// TwinCAT 3 PLC project STS_04
// ProgramVersion: 3.1.4023.0
// libraries:
//   Tc2_Standard, * (Beckhoff Automation GmbH)
//   Tc2_System, * (Beckhoff Automation GmbH)
//   Tc3_Module, * (Beckhoff Automation GmbH)
//   TcUnit, * (www.tcunit.org)
// project tree:
//   DUTs/2. HMI/2.1 HMI Visualization/ dutVisuFeeder.TcDUT, dutVisuMain.TcDUT, dutVisuVBT.TcDUT, dutVisuEjection.TcDUT, dutVisuStacker.TcDUT
//   DUTs/3. Feeder/ FeederMode.TcDUT, FeederSimulation.TcDUT, FeedingState.TcDUT
//   DUTs/1. General State/ GeneralActiveProcessState.TcDUT, GeneralStateCommand.TcDUT, GeneralStateMain.TcDUT
//   DUTs/2. HMI/ HMI.TcDUT
//   DUTs/4. SheetAlignTable/ SheetAlignMode.TcDUT, SheetAlignState.TcDUT
//   DUTs/5. VacuumBeltTable/ VacuumBeltTableMode.TcDUT, VacuumBeltTableState.TcDUT
//   DUTs/6. EjectionGate/ EjectionGateMode.TcDUT, EjectionGateState.TcDUT
//   DUTs/7. StackerBeltTable/ StackerBeltTableMode.TcDUT, StackerBeltTableState.TcDUT
//   GVLs/ GVL.TcGVL, GVL_OOP.TcGVL
//   OOP/0. Program/ MAIN_OOP.TcPOU
//   OOP/1. Physical Buttons/Interface/ I_PB.TcIO
//   OOP/1. Physical Buttons/ PB_NOpen.TcPOU, PB_NClose.TcPOU
//   OOP/2. Physical Sensors/Interface/ I_Sensor.TcIO, O_Sensor.TcIO
//   OOP/2. Physical Sensors/ Sensor_NOpen.TcPOU, Sensor_NClose.TcPOU, Sensor_Trigger.TcPOU
//   OOP/5. Machine/0. Main Machine/ EjectionGate.TcPOU, Feeder.TcPOU, SAT.TcPOU, SBT.TcPOU, VBT.TcPOU
//   OOP/5. Machine/0. Main Machine/Interface/ MachineModule.TcIO
//   OOP/5. Machine/ P_MachineMain.TcPOU, STS.TcPOU
//   / PlcTask.TcTTO
//   POUs/0. FB/ Fb_AnalogToReal_Conversion.TcPOU, Fb_RealToAnalog_Conversion.TcPOU
//   POUs/1.2 Feeder Operation/ Fb_FeederOperation.TcPOU, Fb_FeedingStateCheck.TcPOU, P_Feeder.TcPOU
//   POUs/1.3 Sheet Align Table %28SAT%29/ P_SheetAlignTable.TcPOU (not stored)
//   POUs/1.4 Vacumm Belt Table %28VBT%29/ P_VacummBeltTable.TcPOU (not stored)
//   POUs/1.5 Ejection Gate/ P_EjectionGate.TcPOU
//   POUs/1.6 Stacker Belt Table %28SBT%29/ P_StackerBeltTable.TcPOU (not stored)
//   POUs/1.7 General Movement/ P_AllStateChecker.TcPOU, P_GeneralStateManager.TcPOU
//   POUs/ MAIN.TcPOU, P_Test.TcPOU
//   POUs_Test/ FB_Raw2Analog_Test.TcPOU, PRG_TEST.TcPOU
// real-time tasks:
//   TASK PlcTask: cycle T#10ms, priority 20, ADS port 350

CONFIGURATION STS_04
    RESOURCE PLC ON TwinCAT3
        TASK PlcTask(INTERVAL := T#10ms, PRIORITY := 20);
        PROGRAM MAIN WITH PlcTask : MAIN;
    END_RESOURCE
END_CONFIGURATION

// ---- DUTs/2. HMI/2.1 HMI Visualization/dutVisuFeeder.TcDUT
TYPE dutVisuFeeder :
STRUCT
	(*Values linked to HMI*)
	(*Feeder Operational values*)
	nFormatLength_mm   : INT;
	nSuctionLength_mm  : INT;
	nSheetGap_mm       : INT;
	tSingleSheetTime_s : INT;
	tCompilePostion_s  : INT;
	tDVPIDleOff_s      : INT;
	tDVPStartDelay_s   : INT;
	nMissingSheet      : INT;
	tApproachStop_s    : INT;
	
	(*Sheet Size Adjustment*)
	nSheetSize_mm		: INT;
	bSheetSizeIncrease  : BOOL;
	bSheetSizeDecrease  : BOOL;
	
	(*Feeder Movement setting*)
	bFeederUp			: BOOL;
	bFeederDown         : BOOL;

	(*Start Feeder*)	
	bStartFeeder		: BOOL;
	bStopFeeder			: BOOL;
END_STRUCT
END_TYPE

// ---- DUTs/2. HMI/2.1 HMI Visualization/dutVisuMain.TcDUT
TYPE dutVisuMain :
STRUCT
	(*Main Control*)
	bStartMachine			:BOOL;
	bStopMachine            :BOOL;
	bIncreaseMachineSpeed   :BOOL;
	bDecreaseMachineSpeed   :BOOL;
	                       
	nSheetCountAccepted     :INT;
	nSheetCountRejected     :INT;
	                        
	bSimulationMode         :BOOL;
END_STRUCT
END_TYPE

// ---- DUTs/2. HMI/2.1 HMI Visualization/dutVisuVBT.TcDUT
TYPE dutVisuVBT :
STRUCT
	
	(*Values linked to HMI*)
	(*Vacuum Belt Table Operational values*)
	nVmin_mMin  	: INT;
	nVmax_mMin		: INT;
	tStartDelay_s   : INT;
	tStopDelay_s 	: INT;
	bVisionBypass  	: INT;
	
	(*VBT Jogging*)
	bLeftJog		: BOOL;
	bRightJog  		: BOOL;
	nJogSpeed  		: INT;
	
	(*Fan Volume Control*)
	bFanIncrease	: BOOL;
	bFanDecrease    : BOOL;
	nFanSpeed_pct	: INT;

	(*Start Feeder*)	
	bStartFeeder	: BOOL;
	bStopFeeder		: BOOL;
	
END_STRUCT
END_TYPE

// ---- DUTs/2. HMI/2.1 HMI Visualization/dutVisuEjection.TcDUT
TYPE dutVisuEjection :
STRUCT
	(*Values linked to HMI*)
	(*Rejection Operation*)
	tDetectJamDuration_s	: INT;
	nBrakeDistance_mm		: INT;
	tBrakePulse_ms			: INT;

END_STRUCT
END_TYPE

// ---- DUTs/2. HMI/2.1 HMI Visualization/dutVisuStacker.TcDUT
TYPE dutVisuStacker :
STRUCT
	(*Values linked to HMI*)
	(*Stacker Operational values*)
	tOpenOscillator_s				: INT;
	tCloseJOgger_s      			: int;
	tDownBlas_ms        			: int;
	tDescentPulse_ms    			: int;
	                    			
	(*Stacker Plate Movement*)
	bStackerPlateUp					: BOOL;
	bStackerPlateDown   			: bool;
	                    			
	(*Alignment*)       	
	nAlignmentRation_n				: INT; (*ratio alignment, how many sheets has passed for alignment to trigger*)

	(*Brake Adjustment Control*)
	bIncreaseBrakeSpeedRatio		: BOOL;	
	bDecreaseBrakeSpeedRatio        : BOOL;
	nBrakeSpeedRatio                : INT;
	                                
	bIncreaseBrakeLength            : BOOL;
	bDecreaseBrakeLength            : BOOL;
	nBrakeSpeedLength               : INT;
	                               
	bIncreaseIntersheet             : BOOL;
	bDecreaseIntersheet	            : BOOL;
	nIntersheet                     : INT;

END_STRUCT
END_TYPE

// ---- DUTs/3. Feeder/FeederMode.TcDUT
{attribute 'qualified_only'}
{attribute 'strict'}
TYPE FeederMode :
(
	Mode_Jog		:= 0,
	Mode_Standard	:= 1,
	Mode_Simulation	:= 2
);
END_TYPE

// ---- DUTs/3. Feeder/FeederSimulation.TcDUT
TYPE FeederSimulation :
STRUCT
	i : INT;
END_STRUCT
END_TYPE

// ---- DUTs/3. Feeder/FeedingState.TcDUT
{attribute 'qualified_only'}
{attribute 'strict'}
TYPE FeedingState :
(
	State_Init 					,
	State_AutoStart         	,
	State_AutoHysterisis    	,
	State_AutoStop          	,
	State_AutoTopSensorReached 	,
	State_AutoFinalPosition     ,
	State_AutoBackToInit        ,
	State_Feeding				,
	State_Override				,
	State_Error					,
	State_ManualMoveUp			,
	State_ManualMoveDown    	
 
);
END_TYPE

// ---- DUTs/1. General State/GeneralActiveProcessState.TcDUT
TYPE GeneralActiveProcessState :
STRUCT
	FeederRunning				: BOOL;		 
	FeederStop                  : BOOL;
	FeederError                 : BOOL;
	                         
	SheetAlignTableRunning      : BOOL;
	SheetAlignTableStop         : BOOL;
	SheetAlignTableError        : BOOL;
END_STRUCT
END_TYPE

// ---- DUTs/1. General State/GeneralStateCommand.TcDUT
TYPE GeneralStateCommand :
STRUCT
	
	bStart		:BOOL;
	bStop       :BOOL;
	bOverride   :BOOL;
	bReset		:BOOL;
	
END_STRUCT
END_TYPE

// ---- DUTs/1. General State/GeneralStateMain.TcDUT
{attribute 'qualified_only'}
{attribute 'strict'}
TYPE GeneralStateMain :
(
	
	State_Init			,
	State_Reset         ,
	State_Run	        ,
	State_Stop          ,
	State_ErrorCheck       
);
END_TYPE

// ---- DUTs/2. HMI/HMI.TcDUT
TYPE HMI :
STRUCT
	//-----------------------------Auto----------------------------
	bAuto				:BOOL;
	bStart              :BOOL;
	bStop               :BOOL;
                        
	bFeederManualUp     :BOOL;
	bFeederManualDown   :BOOL;
	(*Visualization*)
	
	FeederOp			: dutVisuFeeder;
	VBTOp               : dutVisuVBT;
	EjectionOP          : dutVisuEjection;
	StackerOP           : dutVisuStacker;
	Main				: dutVisuMain;
	
END_STRUCT
END_TYPE

// ---- DUTs/4. SheetAlignTable/SheetAlignMode.TcDUT
{attribute 'qualified_only'}
{attribute 'strict'}
TYPE SheetAlignMode :
(
	Mode_Standard	:= 0,
	Mode_Manual		:= 1,
	Mode_Simulation	:= 2
	
);
END_TYPE

// ---- DUTs/4. SheetAlignTable/SheetAlignState.TcDUT
{attribute 'qualified_only'}
{attribute 'strict'}
TYPE SheetAlignState :
(
	State_Init 					,
	State_AutoStart         	,
	State_AutoStop          	,
	State_AutoBlowerOn			,
	State_AutoBackToInit        ,
	State_Override				,
	State_Error					
);
END_TYPE

// ---- DUTs/5. VacuumBeltTable/VacuumBeltTableMode.TcDUT
{attribute 'qualified_only'}
{attribute 'strict'}
TYPE VacuumBeltTableMode :
(
	Mode_Standard	:= 0,
	Mode_Manual		:= 1,
	Mode_Simulation	:= 2
	
);
END_TYPE

// ---- DUTs/5. VacuumBeltTable/VacuumBeltTableState.TcDUT
{attribute 'qualified_only'}
{attribute 'strict'}
TYPE VacuumBeltTableState :
(
	State_Init 					,
	State_AutoStart         	,
	State_AutoStop          	,
	State_AutoVacOn				,
	State_VacOff				,
	State_AutoBackToInit        ,
	State_Override				,
	State_Error					
);
END_TYPE

// ---- DUTs/6. EjectionGate/EjectionGateMode.TcDUT
{attribute 'qualified_only'}
{attribute 'strict'}
TYPE EjectionGateMode :
(
	Mode_Standard	:= 0,
	Mode_Manual		:= 1,
	Mode_Simulation	:= 2
	
);
END_TYPE

// ---- DUTs/6. EjectionGate/EjectionGateState.TcDUT
{attribute 'qualified_only'}
{attribute 'strict'}
TYPE EjectionGateState :
(
	State_Init 					,
	State_AutoStart         	,
	State_AutoStop          	,
	State_AutoEjectOn			,
	State_AutoBackToInit        ,
	State_Override				,
	State_Error					
);
END_TYPE

// ---- DUTs/7. StackerBeltTable/StackerBeltTableMode.TcDUT
{attribute 'qualified_only'}
{attribute 'strict'}
TYPE StackerBeltTableMode :
(
	Mode_Standard	:= 0,
	Mode_Manual		:= 1,
	Mode_Simulation	:= 2
	
);
END_TYPE

// ---- DUTs/7. StackerBeltTable/StackerBeltTableState.TcDUT
{attribute 'qualified_only'}
{attribute 'strict'}
TYPE StackerBeltTableState :
(
	State_Init 					,
	State_AutoStart         	,
	State_AutoStop          	,
	State_StackerStart			,
	State_StackerStop	        ,
	State_Override				,
	State_Error					
);
END_TYPE

// ---- GVLs/GVL.TcGVL
{attribute 'qualified_only'}
VAR_GLOBAL
	stHMI 		: HMI;
	stHMIsimul	: HMI;
	bHmiSimulation	: BOOL;
	
	stGSM : GeneralStateCommand; 
END_VAR

// ---- GVLs/GVL_OOP.TcGVL
{attribute 'qualified_only'}
VAR_GLOBAL
	//General Buttons
	(*Governs all things*)
	bStart 	: PB_NOpen; 
	bStop	: PB_NOpen;
	//bStart2 : PB_NClose;
	bEmergencyStop	:PB_NClose;
	
	(*sts component*)
	(*
		sts-feeder
		sts-sat
		sts-vbt
		sts-EjectGate
		sts-Stacker		
	*)
	(*sts-feeder*)
	bBottomHit 		: Sensor_NOpen;
	bTopHit			: Sensor_NOpen;
	bEnableFeeder	: Sensor_Trigger;	
	bUpFeeder		: Sensor_Trigger;
	bResetFeeder	: Sensor_Trigger;
	bDownFeeder     : Sensor_Trigger;
	nFeederTravel   : INT;
	
	(*Modules*)
	stHMI			: HMI;
	
	
	
	fbFeeder		: Feeder(bBottomHit,bTopHit);

	
	fbSTS : STS(bStart,
				bStop,
				bEmergencyStop,
				fbFeeder,
				stHMI);
	
(*OOP Logic*)	
(*
{Sensor Module}
		|
Integrated Into--->{Machine Module}
						|
					Integrated Into ---->{Main Machine}


*)
END_VAR

// ---- OOP/1. Physical Buttons/Interface/I_PB.TcIO
	INTERFACE I_PB

PROPERTY IsPressed : BOOL
//Property of PB when pressed
GET
END_GET
END_PROPERTY

PROPERTY IsReleased : BOOL
//Property of PB when is released
GET
END_GET
END_PROPERTY

END_INTERFACE

// ---- OOP/2. Physical Sensors/Interface/I_Sensor.TcIO
INTERFACE I_Sensor

PROPERTY isActive : BOOL
GET
END_GET
END_PROPERTY

END_INTERFACE

// ---- OOP/2. Physical Sensors/Interface/O_Sensor.TcIO
INTERFACE O_Sensor

PROPERTY isTriggered : BOOL
GET
END_GET
END_PROPERTY

END_INTERFACE

// ---- OOP/5. Machine/0. Main Machine/Interface/MachineModule.TcIO
INTERFACE MachineModule

METHOD Disable : BOOL
VAR_INPUT
END_VAR
END_METHOD

METHOD Enable : BOOL
VAR_INPUT
END_VAR
END_METHOD

METHOD Error : BOOL
VAR_INPUT
END_VAR
END_METHOD

METHOD Override : BOOL
VAR_INPUT
END_VAR
END_METHOD

METHOD Reset : BOOL
VAR_INPUT
END_VAR
END_METHOD

METHOD Start : BOOL
VAR_INPUT
END_VAR
END_METHOD

METHOD PUBLIC StateMachine
VAR_INPUT
END_VAR
END_METHOD

METHOD Stop : BOOL
VAR_INPUT
END_VAR
END_METHOD

END_INTERFACE

// ---- POUs/MAIN.TcPOU
PROGRAM MAIN
VAR
	fb_Test_Conversion : Fb_AnalogToReal_Conversion;
	ntest: LREAL;
	fb_testR2A: Fb_RealToAnalog_Conversion;
	stTestString : STRING :='Added this for 1.0.1';
END_VAR

P_Test();
P_Feeder();
P_SheetAlignTable();
P_VacummBeltTable();
P_EjectionGate();
P_StackerBeltTable();
P_AllStateChecker();
P_GeneralStateManager();
//PRG_TEST();

fb_Test_Conversion(iRawVal:= , iMinVal:=0 , iMaxVal:=180 , lActualVal=>ntest );
fb_testR2A(lActualVal:= , lMinVal:=50 , lMaxVal:=100 , iRawVal=> );

//OOP Test
MAIN_OOP();

END_PROGRAM

// ---- POUs/0. FB/Fb_AnalogToReal_Conversion.TcPOU
FUNCTION_BLOCK Fb_AnalogToReal_Conversion
VAR_INPUT
	iRawVal : UINT;
	iMinVal	: UINT;
	iMaxVal	: UINT;
	
END_VAR
VAR_OUTPUT
	lActualVal	: REAL;				//Actual converted value
	bError		: BOOL;
END_VAR           
VAR               
	lRangeHigh	: REAL := 32676;
	lRawVal 	: REAL;
	lMinVal		: REAL;
	lMaxVal		: REAL;
END_VAR

lRawVal	:=UINT_TO_REAL(iRawVal);
lMinVal	:=UINT_TO_REAL(iMinVal);
lMaxVal	:=UINT_TO_REAL(iMaxVal);

IF iRawVal<=0 THEN
	lActualVal:=0;
END_IF

IF NOT iRawVal>0 AND iRawVal<=lRangeHigh THEN	
	lActualVal := ((lMaxVal-lMinVal)/(lRangeHigh-0))*lRawVal+lMinVal;
	bError:=FALSE;
ELSE
	bError:=TRUE;	
END_IF

METHOD Error_Check : BOOL
VAR_INPUT
END_VAR
END_METHOD

METHOD RawToRealConversion : BOOL
VAR_INPUT
END_VAR
END_METHOD

END_FUNCTION_BLOCK

// ---- POUs/0. FB/Fb_RealToAnalog_Conversion.TcPOU
FUNCTION_BLOCK Fb_RealToAnalog_Conversion
VAR_INPUT
	lActualVal	: REAL;
	lMinVal		: REAL;
	lMaxVal		: REAL;
	
END_VAR
VAR_OUTPUT
	iRawVal	: UINT;					//Raw converted sensor values
END_VAR           
VAR               
	lRangeHigh	: REAL := 32676;
	lRawVal : REAL;

END_VAR


IF lActualVal <=0 THEN
	iRawVal:=0;
END_IF

IF lActualVal>0 THEN
	lRawVal:=(lActualVal-lMinVal)*((lRangeHigh-0)/(lMaxVal-lMinVal));
END_IF

END_FUNCTION_BLOCK

// ---- POUs/P_Test.TcPOU
PROGRAM P_Test
VAR
	
nAngle : LREAL;
nAngle_decimal : int;
nAngle_Final : LREAL;
sWriteFromHMI : STRING;
sWriteToHMI : STRING:='This Is From PLC';
b_HMI_StartLine : BOOL;
b_HMI_StopLine : BOOL;
bStartTrig: R_TRIG;
bStopTrig: R_TRIG;

bSpeedInc		:BOOL;
bSpeedDecrease  :BOOL;
stStatus		:STRING;
// State
n : INT;
END_VAR


bStartTrig(CLK:=b_HMI_StartLine , Q=> );
bStopTrig(CLK:=b_HMI_StopLine , Q=> );

IF ( stStatus='' OR stStatus='Stopped') 
	AND bStartTrig.Q THEN
	stStatus:='Started';

END_IF

IF stStatus='Started' AND bStopTrig.Q THEN
	stStatus:='Stopped';
	nAngle :=0;
END_IF

IF  stStatus='Started' THEN
	
	IF nAngle<180 THEN
		nAngle :=nAngle+0.01;
	END_IF
	//nAngle_decimal:=find((LREAL_TO_STRING(nAngle)),'.');
		
	IF nAngle>=180 THEN
		nAngle :=0;
	END_IF
END_IF
nAngle_Final :=LREAL_TO_UINT(STRING_TO_LREAL(left((LREAL_TO_STRING(nAngle)),((find((LREAL_TO_STRING(nAngle)),'.'))+2))));

END_PROGRAM

// ---- POUs/1.2 Feeder Operation/P_Feeder.TcPOU
PROGRAM P_Feeder
VAR
	bStartFeeder : BOOL;
	bFeederOK: BOOL;
	//dut_FeedingState : FeedingState;
	fbFb_FeedingStateCheck: Fb_FeedingStateCheck;	
//-----------------------------------Feeder Mode -------------------------//
	iFeederMode : INT;	
	bGoCounter, bSetCounter AT %Q*:BOOL;
	wFrequencyValue, wTargetCounterValue, wSetCounterValue AT %Q*:WORD;
	wCounterValue AT %I*:WORD;
	nState, nCntCycle:UDINT;
	bStart:BOOL;
	wFrequencyValue_Test:WORD:=200;
	nPrevValue			:WORD;
	wTargetCounterValue_Test:WORD:=180;
	bHitTop : BOOL;
	bHitBottom : BOOL;
	bTargetDistanceHitUP	: BOOL;
	bTargetDistanceHitDown	: BOOL;

//------------------------------------CASE-------------------------------//
	ifeedercase : INT;

(* For reference
	State_Init 					:= 1,
	State_AutoStart         	:= 2,
	State_AutoHysterisis    	:= 3,
	State_AutoStop          	:= 4,
	State_AutoTopSensorReached 	:= 5,
	State_AutoFinalPosition     := 6,
	State_AutoBackToInit        := 7,
	State_Feeding				:= 8,
	State_Override				:= 9,
	State_Error					:= 10,
	State_ManualMoveUp			:= 11,
	State_ManualMoveDown    	:= 12
*)	
//-------------------------Simulated Values-----------------------------//
nCurrentValue 	: DWORD;
nTargetValue	: DWORD;
	
END_VAR
VAR_INPUT
	bStartCommand : BOOL;
END_VAR

IF GVL.bHmiSimulation THEN
	GVL.stHMIsimul:=GVL.stHMI;
	iFeederMode:=FeederMode.Mode_Simulation;
END_IF 
IF NOT GVL.bHmiSimulation THEN
	GVL.stHMI:=GVL.stHMI;
	iFeederMode:=FeederMode.Mode_Standard;
END_IF

CASE ifeedercase OF

FeedingState.State_Init 			:	//Awaiting for command   
	IF GVL.stHMI.bAuto  THEN
		ifeedercase:=FeedingState.State_AutoStart;
	END_IF
	IF GVL.stHMI.bFeederManualDown THEN
		ifeedercase:=FeedingState.State_ManualMoveDown;	
	END_IF
	IF GVL.stHMI.bFeederManualUp THEN
		ifeedercase:=FeedingState.State_ManualMoveUp;
	END_IF	
	IF NOT (iFeederMode=FeederMode.Mode_Simulation) THEN // go back to init
		iFeederCase:=FeedingState.State_Init;
		wTargetCounterValue:=0;
		nPrevValue:=0;	
		bHitTop:=FALSE;	
		bHitBottom:=FALSE;
		bTargetDistanceHitUp:=FALSE;
		bTargetDistanceHitDown:=FALSE;
		nState:=0;
	END_IF
	
FeedingState.State_AutoStart            : 	//Start 

	IF NOT bStartFeeder THEN
		ifeedercase:= FeedingState.State_AutoBackToInit;
	END_IF
	IF GVL.bHmiSimulation THEN
		//Adding Feeder movement simulation
		;
	END_IF
FeedingState.State_AutoHysterisis       : 
FeedingState.State_AutoStop             : 
FeedingState.State_AutoTopSensorReached :	
FeedingState.State_AutoFinalPosition    : 
FeedingState.State_AutoBackToInit       : 
FeedingState.State_Feeding				:        
FeedingState.State_Override				:       
FeedingState.State_Error				:	
     
FeedingState.State_ManualMoveUp			:
	IF iFeederMode=FeederMode.Mode_Simulation THEN
		CASE nState OF
				0: //Check ongoing or Initial Start
					IF gvl.stHMI.bFeederManualUp THEN
						IF NOT (bHitTop OR bTargetDistanceHitUp) THEN
							IF nPrevValue=0 
							AND wTargetCounterValue=0 THEN // Coming from initialization
								nState:=20;
							END_IF
							IF wTargetCounterValue>nPrevValue THEN //Continuation
								nPrevValue:=wTargetCounterValue;
								nState:=20;
							END_IF
						ELSE
							nState:=0;
							nPrevValue:=wTargetCounterValue;
						END_IF
					END_IF	
					
				20://Increment and making sure previous values are recorded.			
							IF (wTargetCounterValue>nPrevValue) THEN
								nState:=30;
							END_IF
							IF (wTargetCounterValue=nPrevValue) THEN
								wTargetCounterValue:=wTargetCounterValue+1;
								nState:=20;
							END_IF

				30:	//Check if reached target or not
					IF wTargetCounterValue < wTargetCounterValue_Test THEN //not reached
						nstate:=0;
					END_IF
					IF wTargetCounterValue >= wTargetCounterValue_Test OR bHitTop THEN // Reached sensor top or movement set
						nState:=40;
					END_IF
				40:	
					nState:=0;
					bTargetDistanceHitUp:=TRUE;
					bFeederOK :=TRUE;
					
				
		END_CASE
	END_IF
	IF iFeederMode=FeederMode.Mode_Jog THEN
		;
	END_IF
	ifeedercase:= FeedingState.State_Init;
	
FeedingState.State_ManualMoveDown		:
	IF iFeederMode=FeederMode.Mode_Simulation THEN
		CASE nState OF
				0: //Check ongoing or Initial Start
					IF gvl.stHMI.bFeederManualDown THEN
						IF NOT (bHitBottom OR bTargetDistanceHitDown) THEN
							IF nPrevValue=0 
							AND wTargetCounterValue=0 THEN // Coming from initialization
								nState:=20;
							END_IF
							IF wTargetCounterValue>nPrevValue THEN //Continuation
								nPrevValue:=wTargetCounterValue;
								nState:=20;
							END_IF
						ELSE
							nState:=0;
							nPrevValue:=wTargetCounterValue;
						END_IF
					END_IF	
					
				20://Increment and making sure previous values are recorded.			
							IF (wTargetCounterValue>nPrevValue) THEN
								nState:=30;
							END_IF
							IF (wTargetCounterValue=nPrevValue) THEN
								wTargetCounterValue:=wTargetCounterValue+1;
								nState:=20;
							END_IF

				30:	//Check if reached target or not
					IF wTargetCounterValue < wTargetCounterValue_Test THEN //not reached
						nstate:=0;
					END_IF
					IF wTargetCounterValue >= wTargetCounterValue_Test OR bHitTop THEN // Reached sensor top or movement set
						nState:=40;
					END_IF
				40:	
					nState:=0;
					bTargetDistanceHitDown:=TRUE;
				
		END_CASE
	END_IF
	IF iFeederMode=FeederMode.Mode_Jog THEN
		;
	END_IF
	ifeedercase:= FeedingState.State_Init;
	

END_CASE

END_PROGRAM

// ---- POUs/1.2 Feeder Operation/Fb_FeedingStateCheck.TcPOU
FUNCTION_BLOCK Fb_FeedingStateCheck
VAR_INPUT
	dut_FeedingState : FeedingState;
END_VAR
VAR_OUTPUT
	iReadableFeedingState : INT; // number which represent the state
END_VAR
VAR
	iBareNum : INT; // number we use to cycle through the FeedingState
	iLastFeedingState : FeedingState;
	
	nCaseNumberCycler : INT;
END_VAR

CASE nCaseNumberCycler OF
0: //Check if number is 0 or not. As 0 would represent initialized state
	//Also check whether it is there are any state changes or not
	IF (dut_FeedingState = iLastFeedingState ) THEN
		nCaseNumberCycler:=0;
	ELSE
		nCaseNumberCycler:=10;
	END_IF
	
10: //Cycling
	FOR iBareNum:=0 TO 11 BY 1 DO
		IF iBareNum < dut_FeedingState THEN
			iBareNum:=iBareNum+1;
		END_IF
		IF iBareNum > dut_FeedingState THEN
			iBareNum:=iBareNum-1;
		END_IF
		
	END_FOR
nCaseNumberCycler:=50;
50:	
nCaseNumberCycler:=0;
END_CASE

END_FUNCTION_BLOCK

// ---- POUs/1.5 Ejection Gate/P_EjectionGate.TcPOU
PROGRAM P_EjectionGate
VAR
		(*Initialization*)
	bEJ_OK		: BOOL;
	bError		: BOOL;
	bStart		: BOOL;
	bStop		: BOOL;
	(*Process*)
	bEjEnable 	: BOOL;
	bEjectOn	: BOOL;
	bEjectOff	: BOOL;
	bOverride	: BOOL;
	(*Ejection Gate Specific Process*)
	bSheetStuck		: BOOL;
	bSheetPresence		: BOOL;
	nSheetCount		: INT;
	FB_SheetCount_Trig	: R_TRIG;
	tSheetStuck_s	: TIME :=T#5S ;
	
	
	//-----------------------------------------(*Case*)-----------------------------------------------------
	
	(* Reference for VBT

	State_Init 					,
	State_AutoStart         	,
	State_AutoStop          	,
	State_AutoEjectOn			,
	State_AutoBackToInit        ,
	State_Override				,
	State_Error			
	*)	
	
	asd: R_TRIG;
	FbSheetStuckCheck: TON;
END_VAR
VAR_INPUT
	bStartCommand : BOOL;
END_VAR
VAR_OUTPUT
	iEJcase : INT;
END_VAR

CASE iEJcase OF
EjectionGateState.State_Init			:	

	IF (bEJ_OK AND bStartCommand)  
	AND NOT bError THEN
		iEJcase:= EjectionGateState.State_AutoStart;
	END_IF 
	IF bError THEN
		iEJcase:= EjectionGateState.State_Error;
	END_IF

   
EjectionGateState.State_AutoStart     	:
	IF bStop THEN
		iEJcase:= EjectionGateState.State_AutoStop;
	ELSE
		iEJcase :=EjectionGateState.State_AutoEjectOn;
	END_IF


EjectionGateState.State_AutoStop      	:
	iEJcase:= EjectionGateState.State_AutoBackToInit;


EjectionGateState.State_AutoEjectOn	  	:
	(*Insert business logic here*)
	(*Ejection*)
	IF P_VacummBeltTable.bBadSheetSignal THEN
		bEjectOn :=TRUE;
	END_IF // Need to add business logic to count for speed/time on-site.
	
	(*Sheet Counting*)
	FB_SheetCount_Trig(CLK:= bSheetPresence, Q=> );
	IF FB_SheetCount_Trig.Q THEN
		nSheetCount:=nSheetCount+1;
	END_IF
	FbSheetStuckCheck(IN:=bSheetPresence , PT:=tSheetStuck_s , Q=> , ET=> );
	IF FbSheetStuckCheck.Q THEN
		bSheetStuck:=TRUE;
		iEJcase:= EjectionGateState.State_Error;
	END_IF


EjectionGateState.State_AutoBackToInit	:
	iEJcase:= EjectionGateState.State_Init;


EjectionGateState.State_Override		:   
	;


EjectionGateState.State_Error			:     
	IF bError THEN
		iEJcase:= EjectionGateState.State_AutoBackToInit;
	END_IF

END_CASE

END_PROGRAM

// ---- POUs/1.7 General Movement/P_AllStateChecker.TcPOU
PROGRAM P_AllStateChecker
VAR
	(*
		Author - Gideon Jgordon (GJ)
		Changes 
		-(GJ) stGSM moved here
	*)	
	bAllOk : BOOL;	// All OK process
	//bSAT_OK: BOOL;  //SAT Process OK
END_VAR


IF P_GeneralStateManager.nStateGeneral =GeneralStateMain.State_ErrorCheck THEN
	gvl.stGSM.bStop			:=TRUE;
	gvl.stGSM.bOverride		:=FALSE;
	gvl.stGSM.bStart		:=FALSE;
	gvl.stGSM.bReset		:=TRUE;	
END_IF

IF P_GeneralStateManager.nStateGeneral =GeneralStateMain.State_Init THEN
	gvl.stGSM.bStop		   :=TRUE;
	gvl.stGSM.bOverride	   :=TRUE;
	gvl.stGSM.bStart	   :=FALSE;
	gvl.stGSM.bReset	   :=FALSE;	
END_IF

IF P_GeneralStateManager.nStateGeneral =GeneralStateMain.State_Reset THEN
	gvl.stGSM.bStop		   :=TRUE;
	gvl.stGSM.bOverride	   :=FALSE;
	gvl.stGSM.bStart	   :=FALSE;
	gvl.stGSM.bReset	   :=TRUE;	
END_IF

IF P_GeneralStateManager.nStateGeneral =GeneralStateMain.State_Run THEN
	gvl.stGSM.bStop		   :=TRUE;
	gvl.stGSM.bOverride	   :=FALSE;
	gvl.stGSM.bStart	   :=FALSE;
	gvl.stGSM.bReset	   :=FALSE;
END_IF

IF P_GeneralStateManager.nStateGeneral =GeneralStateMain.State_Stop THEN
	gvl.stGSM.bStop		   :=TRUE;
	gvl.stGSM.bOverride	   :=FALSE;
	gvl.stGSM.bStart	   :=FALSE;
	gvl.stGSM.bReset	   :=FALSE;
END_IF

IF  	P_Feeder.bFeederOK 
	AND P_SheetAlignTable.bSAT_OK 
	AND P_VacummBeltTable.bVBT_OK
	AND P_EjectionGate.bEJ_OK
	AND P_StackerBeltTable.bSBT_OK		THEN
	bAllok:=TRUE;
ELSE
	bAllok:=FALSE;	
END_IF

END_PROGRAM

// ---- POUs/1.7 General Movement/P_GeneralStateManager.TcPOU
PROGRAM P_GeneralStateManager
VAR
	(*
		Author - Gideon Jgordon (GJ)
		Changes 
		-(GJ) Added to govern the General State of the STS04 Machine 
		-(GJ) stGSM moved to P_AllStateChecker to make it cleaner
	*)	
	nStateGeneral : INT;
	bValuesResetDone: BOOL;
END_VAR

CASE nStateGeneral OF

GeneralStateMain.State_Init				: //Initialize all the state

	IF gvl.stHMI.bStart THEN
		nStateGeneral:= GeneralStateMain.State_Reset;
		ELSE
		nStateGeneral:=	GeneralStateMain.State_Init;
	END_IF	
	
GeneralStateMain.State_Reset			: // Reset behaviour and values befor we proceed to go into Run Mode

	//Adding reset below here
	IF (bValuesResetDone AND P_AllStateChecker.bAllOk) THEN
		nStateGeneral:=GeneralStateMain.State_Run;
		gvl.stGSM.bStart	:=TRUE;
	END_IF
	IF NOT (bValuesResetDone AND P_AllStateChecker.bAllOk) THEN
		nStateGeneral:=GeneralStateMain.State_Init;
	END_IF
	
GeneralStateMain.State_Run              : // Governs the Process during run

	IF NOT P_AllStateChecker.bAllOk THEN
		gvl.stGSM.bStart	:=FALSE;
	END_IF
	IF gvl.stHMI.bStop THEN
		nStateGeneral:= GeneralStateMain.State_Stop;
		gvl.stGSM.bStart	:=FALSE;
	END_IF
	
GeneralStateMain.State_Stop             : //Stop via HMI or Error

	nStateGeneral:= GeneralStateMain.State_Init;
	
GeneralStateMain.State_ErrorCheck       :

	
	
END_CASE

END_PROGRAM

// ---- OOP/0. Program/MAIN_OOP.TcPOU
PROGRAM MAIN_OOP
VAR
	bStartButton : PB_NOpen;
	bStopButton :PB_NOpen;
	bEstopButton : PB_NClose;
	bProcessStart : BOOL;
	bProcessError : BOOL;
	bProcessOverride : BOOL;
	
	//Feeder
	bStartFeeder		: BOOL;
	bStopFeeder			: BOOL;
	bFeederError        : BOOL;
	                   
	bFeederAuto         : BOOL;
	bFeederUpAuto       : BOOL;
	bFeederDownAuto     : BOOL;
	                   
	bFeederManual       : BOOL;
	bFeederUpManual     : BOOL;
	bFeederDownManual   : BOOL;
	
	bFeederAtPos		: BOOL;
	
	// SAT
	
	
END_VAR

IF bStartButton.IsPressed AND bStopButton.IsPressed THEN
	bStartFeeder:=TRUE;
END_IF
IF bStopButton.IsPressed AND bStartButton.IsPressed THEN
	bStopFeeder :=FALSE;
END_IF

P_MachineMain();

END_PROGRAM

// ---- OOP/1. Physical Buttons/PB_NOpen.TcPOU
FUNCTION_BLOCK PB_NOpen IMPLEMENTS I_PB
VAR
	bInput AT %I* :BOOL;
	
END_VAR

PROPERTY IsPressed : BOOL
//Property of PB when pressed
GET
VAR
	//Giving the properties of bInputSensor to isPressed
END_VAR
IsPressed := bInput;
END_GET
END_PROPERTY

PROPERTY IsReleased : BOOL
//Property of PB when PBNOpen is released
GET
VAR
	//Giving the properties of bInputSensor to isPressed
END_VAR
IsReleased := NOT bInput;
END_GET
END_PROPERTY

END_FUNCTION_BLOCK

// ---- OOP/1. Physical Buttons/PB_NClose.TcPOU
FUNCTION_BLOCK PB_NClose IMPLEMENTS I_PB
VAR
	bInput AT %I* :BOOL;
	
END_VAR

PROPERTY IsPressed : BOOL
// Property of PB button when it is pressed but for normally close
GET
IsPressed := NOT bInput;
END_GET
END_PROPERTY

PROPERTY IsReleased : BOOL
// Property of PB button when it is Released State but for normally close
GET
IsReleased := bInput;
END_GET
END_PROPERTY

END_FUNCTION_BLOCK

// ---- OOP/5. Machine/P_MachineMain.TcPOU
PROGRAM P_MachineMain
VAR
	
END_VAR

GVL_OOP.fbFeeder();
GVL_OOP.fbSTS();

END_PROGRAM

// ---- OOP/5. Machine/STS.TcPOU
FUNCTION_BLOCK STS
VAR
	bStart	: I_PB; // ref this to NO How to reference this as NO or NC????
	//bStart2	: I_PB;
	bStop	: I_PB; // ref this of NO
	bEmergency	: I_PB; // ref this to NC
	Feeder : MachineModule; // ref this to MachineModule
	
	// HMI here
	STS_Hmi : HMI;	
	
	

END_VAR

IF bStart.IsPressed AND bStop.IsReleased THEN
	Feeder.Enable();
END_IF

IF bStart.IsReleased AND bStop.IsPressed THEN
	Feeder.Disable();
END_IF

IF bEmergency.IsPressed THEN
	Feeder.Disable();
END_IF

METHOD FB_init : BOOL
VAR_INPUT
	bInitRetains : BOOL; // if TRUE, the retain variables are initialized (warm start / cold start)
	bInCopyCode : BOOL;  // if TRUE, the instance afterwards gets moved into the copy code (online change)
	
// Parsing it so that the STS declared need to have 4 arguments	
	bStart	: I_PB; // ref this to NO How to reference this as NO or NC????
	bStop	: I_PB; // ref this of NO
	bEmergency	: I_PB; // ref this to NC
	
	//Machine Modules
	Feeder : MachineModule; // ref this to MachineModule
	STS_Hmi : HMI;	
	
END_VAR
THIS^.bStart			:= bStart;
THIS^.bStop			:= bStop;
THIS^.bEmergency	    := bEmergency;
THIS^.Feeder          := Feeder;
THIS^.STS_Hmi         := STS_Hmi;
END_METHOD

END_FUNCTION_BLOCK

// ---- OOP/5. Machine/0. Main Machine/Feeder.TcPOU
FUNCTION_BLOCK Feeder IMPLEMENTS MachineModule
VAR
	(*General Movement Trigger*)
	bEnable			: BOOL;
	bDisable        : BOOL;
	bError          : BOOL;
	bOverride       : BOOL;
	bSimulation     : BOOL;
	bStart          : BOOL;
	bStop           : BOOL;
	
	(*Sensor Specific Trigger*)
	bBottomHit 		: I_Sensor;
	bTopHit			: I_Sensor;
	(*Internal Variable*)
	nMovement 		: INT;
	nmovetest		: INT;
	(*Fedder*)
	bFeederPlateInPos	: BOOL;

END_VAR

(*Business Logic here*)

IF 	bEnable 
	AND NOT (bError)
	AND nMovement<1500 THEN
	
	nMovement := nMovement+1;
	bStop:=FALSE; (*Could use this thing in another module*)
	
END_IF

IF nMovement=1500 THEN
	bStop:=TRUE;
END_IF

METHOD Disable : BOOL 
VAR_INPUT
END_VAR
bEnable:=FALSE;
END_METHOD

METHOD Enable : BOOL
VAR_INPUT
END_VAR
bEnable:=TRUE;
bDisable:=FALSE;
END_METHOD

METHOD Error : BOOL
VAR_INPUT
END_VAR
bEnable:=FALSE;
END_METHOD

METHOD FB_init : BOOL
VAR_INPUT
	bInitRetains : BOOL; // if TRUE, the retain variables are initialized (warm start / cold start)
	bInCopyCode : BOOL;  // if TRUE, the instance afterwards gets moved into the copy code (online change)
	bBottomHit 		: I_Sensor;
	bTopHit			: I_Sensor;
END_VAR
THIS^.bBottomHit	:= bBottomHit;
THIS^.bTopHit		:= bTopHit;
END_METHOD

METHOD Override : BOOL
VAR_INPUT
END_VAR
END_METHOD

METHOD Reset : BOOL
VAR_INPUT
END_VAR
END_METHOD

METHOD Start : BOOL
VAR_INPUT
END_VAR
END_METHOD

METHOD PUBLIC StateMachine
VAR_INPUT

END_VAR
IF bEnable THEN
	nmovetest:=nmovetest+1;	
	ELSE
		
	nmovetest:=0;
END_IF
END_METHOD

METHOD Stop : BOOL
VAR_INPUT
END_VAR
END_METHOD

END_FUNCTION_BLOCK

// ---- OOP/5. Machine/0. Main Machine/SAT.TcPOU
FUNCTION_BLOCK SAT IMPLEMENTS MachineModule
VAR
	bEnable			: BOOL;
	bDisable        : BOOL;
	bError          : BOOL;
	bOverride       : BOOL;
	bSimulation     : BOOL;
	bStart          : BOOL;
	bStop           : BOOL;
END_VAR

// This is the core module needed that we are creating for our STS and contains everything related to the STS

// To be added
(*
FEEDER

SAT

VBT

EJECT

GATE

SBT

*)

METHOD Disable : BOOL
VAR_INPUT
END_VAR
bEnable:=FALSE;
END_METHOD

METHOD Enable : BOOL
VAR_INPUT
END_VAR
bEnable:=TRUE;
bDisable:=False;
END_METHOD

METHOD Error : BOOL
VAR_INPUT
END_VAR
bEnable:=FALSE;
END_METHOD

METHOD Override : BOOL
VAR_INPUT
END_VAR
END_METHOD

METHOD Reset : BOOL
VAR_INPUT
END_VAR
END_METHOD

METHOD Start : BOOL
VAR_INPUT
END_VAR
END_METHOD

METHOD PUBLIC StateMachine
VAR_INPUT
END_VAR
END_METHOD

METHOD Stop : BOOL
VAR_INPUT
END_VAR
END_METHOD

END_FUNCTION_BLOCK

// ---- OOP/5. Machine/0. Main Machine/VBT.TcPOU
FUNCTION_BLOCK VBT IMPLEMENTS MachineModule
VAR
	bEnable			: BOOL;
	bDisable        : BOOL;
	bError          : BOOL;
	bOverride       : BOOL;
	bSimulation     : BOOL;
	bStart          : BOOL;
	bStop           : BOOL;
END_VAR

// This is the core module needed that we are creating for our STS and contains everything related to the STS

// To be added
(*
FEEDER

SAT

VBT

EJECT

GATE

SBT

*)

METHOD Disable : BOOL
VAR_INPUT
END_VAR
bEnable:=FALSE;
END_METHOD

METHOD Enable : BOOL
VAR_INPUT
END_VAR
bEnable:=TRUE;
bDisable:=False;
END_METHOD

METHOD Error : BOOL
VAR_INPUT
END_VAR
bEnable:=FALSE;
END_METHOD

METHOD Override : BOOL
VAR_INPUT
END_VAR
END_METHOD

METHOD Start : BOOL
VAR_INPUT
END_VAR
END_METHOD

METHOD PUBLIC StateMachine
VAR_INPUT
END_VAR
END_METHOD

METHOD Stop : BOOL
VAR_INPUT
END_VAR
END_METHOD

END_FUNCTION_BLOCK

// ---- OOP/2. Physical Sensors/Sensor_NOpen.TcPOU
FUNCTION_BLOCK Sensor_NOpen IMPLEMENTS I_Sensor
VAR
	bInput AT %I* : BOOL;
END_VAR

PROPERTY isActive : BOOL
GET
isActive:=bInput;
END_GET
END_PROPERTY

PROPERTY notActive : BOOL
GET
notActive:= NOT bInput;
END_GET
END_PROPERTY

END_FUNCTION_BLOCK

// ---- OOP/2. Physical Sensors/Sensor_Trigger.TcPOU
FUNCTION_BLOCK Sensor_Trigger implements O_Sensor
VAR
	bOutput AT %Q* : BOOL;
END_VAR

PROPERTY isTriggered : BOOL
GET
isTriggered:=bOutput;
END_GET
END_PROPERTY

END_FUNCTION_BLOCK

// ---- OOP/2. Physical Sensors/Sensor_NClose.TcPOU
FUNCTION_BLOCK Sensor_NClose IMPLEMENTS I_Sensor
VAR
	bInput AT %I* : BOOL;
END_VAR

PROPERTY isActive : BOOL
GET
isActive:= not bInput;
END_GET
END_PROPERTY

PROPERTY notActive : BOOL
GET
isActive := bInput;
END_GET
END_PROPERTY

END_FUNCTION_BLOCK

// ---- OOP/5. Machine/0. Main Machine/EjectionGate.TcPOU
FUNCTION_BLOCK EjectionGate IMPLEMENTS MachineModule
VAR
	bEnable			: BOOL;
	bDisable        : BOOL;
	bError          : BOOL;
	bOverride       : BOOL;
	bSimulation     : BOOL;
	bStart          : BOOL;
	bStop           : BOOL;
END_VAR

// This is the core module needed that we are creating for our STS and contains everything related to the STS

// To be added
(*
FEEDER

SAT

VBT

EJECT

GATE

SBT

*)

METHOD Disable : BOOL
VAR_INPUT
END_VAR
bEnable:=FALSE;
END_METHOD

METHOD Enable : BOOL
VAR_INPUT
END_VAR
bEnable:=TRUE;
bDisable:=False;
END_METHOD

METHOD Error : BOOL
VAR_INPUT
END_VAR
bEnable:=FALSE;
END_METHOD

METHOD Override : BOOL
VAR_INPUT
END_VAR
END_METHOD

METHOD Reset : BOOL
VAR_INPUT
END_VAR
END_METHOD

METHOD Start : BOOL
VAR_INPUT
END_VAR
END_METHOD

METHOD PUBLIC StateMachine
VAR_INPUT
END_VAR
END_METHOD

METHOD Stop : BOOL
VAR_INPUT
END_VAR
END_METHOD

END_FUNCTION_BLOCK

// ---- OOP/5. Machine/0. Main Machine/SBT.TcPOU
FUNCTION_BLOCK SBT IMPLEMENTS MachineModule
VAR
	bEnable			: BOOL;
	bDisable        : BOOL;
	bError          : BOOL;
	bOverride       : BOOL;
	bSimulation     : BOOL;
	bStart          : BOOL;
	bStop           : BOOL;
END_VAR

// This is the core module needed that we are creating for our STS and contains everything related to the STS

// To be added
(*
FEEDER

SAT

VBT

EJECT

GATE

SBT

*)

METHOD Disable : BOOL
VAR_INPUT
END_VAR
bEnable:=FALSE;
END_METHOD

METHOD Enable : BOOL
VAR_INPUT
END_VAR
bEnable:=TRUE;
bDisable:=False;
END_METHOD

METHOD Error : BOOL
VAR_INPUT
END_VAR
bEnable:=FALSE;
END_METHOD

METHOD Override : BOOL
VAR_INPUT
END_VAR
END_METHOD

METHOD Reset : BOOL
VAR_INPUT
END_VAR
END_METHOD

METHOD Start : BOOL
VAR_INPUT
END_VAR
END_METHOD

METHOD PUBLIC StateMachine
VAR_INPUT
END_VAR
END_METHOD

METHOD Stop : BOOL
VAR_INPUT
END_VAR
END_METHOD

END_FUNCTION_BLOCK

// ---- POUs/1.2 Feeder Operation/Fb_FeederOperation.TcPOU
FUNCTION_BLOCK Fb_FeederOperation
VAR_INPUT
	nModeSelector	: FeederMode;
	bEnable         : BOOL;
END_VAR
VAR_OUTPUT
	bJogFwd         : BOOL;
	bJogRev         : BOOL;
END_VAR
VAR
END_VAR

;

END_FUNCTION_BLOCK

// ---- POUs_Test/FB_Raw2Analog_Test.TcPOU
FUNCTION_BLOCK FB_Raw2Analog_Test extends FB_TestSuite
VAR
END_VAR

TestRawVal2RealValConversion();

METHOD PRIVATE TestRawVal2RealValConversion EXTENDS FB_TestSuite
VAR
	Fb_Raw2Analog	: Fb_AnalogToReal_Conversion;
	nReal : REAL;
	bError : BOOL;
END_VAR
TEST('TestRawVal2RealValConversion');

//Value 1 test
Fb_Raw2Analog(iRawVal:=32676 , iMinVal:=0 , iMaxVal:=100 , lActualVal=> , bError =>bError );
AssertEquals_REAL(	Expected :=100,
					Actual:=Fb_Raw2Analog.lActualVal,
					Delta:= 0.5,
					Message:='Expected Delta < 0.5');

TEST_FINISHED();
END_METHOD

END_FUNCTION_BLOCK

// ---- POUs_Test/PRG_TEST.TcPOU
PROGRAM PRG_TEST
VAR
	fbAnalog2Real_TEST :FB_Raw2Analog_Test;
END_VAR

 TcUnit.RUN();

END_PROGRAM
